// Implicitly generated code : DO NOT EDIT
FUNCTION CheckRangeSigned : DINT
VAR_INPUT
	value, lower, upper: DINT;
END_VAR
VAR
    sMessageLow   : STRING := 'CheckRangeSigned: Value too low (%d)';
    sMessageHigh  : STRING := 'CheckRangeSigned: Value too high (%d)';
END_VAR

// Implicitly generated code : Only an Implementation suggestion
{noflow}
IF (value < lower) THEN
	CheckRangeSigned := lower;
    // Log message
    ADSLOGDINT(msgCtrlMask := ADSLOG_MSGTYPE_WARN,
               msgFmtStr   := sMessageLow,
               dintArg     := value);
ELSIF(value > upper) THEN
	CheckRangeSigned := upper;
	// Log message
    ADSLOGDINT(msgCtrlMask := ADSLOG_MSGTYPE_WARN,
               msgFmtStr   := sMessageHigh,
               dintArg     := value);
ELSE
	CheckRangeSigned := value;
END_IF
{flow}

END_FUNCTION

(* stored: Version 1.1.0.1, ProductVersion 3.1.4024.11
   POU CheckRangeSigned: Id {4d4c37aa-cb3b-4242-bc05-138b434dab29}, SpecialFunc CheckRangeSigned *)
